PROGRAM MAIN
VAR
	arrInputPNP AT %I* : ARRAY[0..GVL.cuiNrChannel] OF BOOL;
	arrInputNPN	AT %I* : ARRAY[0..GVL.cuiNrChannel] OF BOOL;
END_VAR

arrInputPNP;
arrInputNPN;

END_PROGRAM

(* stored: Version 1.1.0.1, ProductVersion 3.1.4024.6
   POU MAIN: Id {4d55c260-25ae-4664-9203-47957f836f1e}, SpecialFunc None *)
